VISUALIZATION VISU_DummyState  // 2x2
END_VISUALIZATION

(* stored: Version 1.1.0.1, ProductVersion 3.1.4024.11
   Visu VISU_DummyState: Id {4109fb55-7800-4eb2-80b6-fa117aaf59fc} *)
